TYPE dutResponse :
STRUCT
END_STRUCT
END_TYPE

(* stored: Version 1.1.0.1, ProductVersion 3.1.4024.12
   DUT dutResponse: Id {8b5ea8bb-766a-46e8-93f9-756088c40349} *)
